Staubli VAL3: cartesianSpace.pjx

Parameters version=s7.9.1 stackSize=5000 millimeterUnit=true
Data file=cartesianSpace.dtx
Type name=CartesianPos path=./CartesianPos/CartesianPos.pjx
Type name=CartesianVel path=./CartesianVel/CartesianVel.pjx
Type name=CartesianAccel path=./CartesianAccel/CartesianAccel.pjx
Type name=CartesianForce path=./CartesianForce/CartesianForce.pjx
